// ---- DUTs/IO/Topology/Beckhoff_EPP1xxxEK1122_5ECABF39.TcDUT
{attribute 'GeneratedUsingTerminal: EK1122-0000-0018'}
{attribute addProperty BoxType "EK1122-0000-0018"}
{attribute addProperty Id "Beckhoff_EPP1xxxsub_EK1100EK1100_1FC0878B2A_0001_EPP1004_0061_0016EPP1004_D135F8DB8A_0002_EPP1008_0001_0016EPP1008_78E8D3DD12A_0003_EPP1008_0001_0017EPP1008_78E8D3DD12A_0004_EPP1008_0002_0016EPP1008_78E8D3DD12A_0005_EPP1008_0002_0017EPP1008_78E8D3DD12A_0006_EPP1008_0022_0016EPP1008_78E8D3DD12A_0007_EPP1018_0001_0016EPP1018_78E8D3DD12A_0008_EPP1018_0001_0017EPP1018_78E8D3DD12A_0009_EPP1018_0002_0016EPP1018_78E8D3DD12A_0010_EPP1018_0002_0017EPP1018_78E8D3DD12A_0011_EPP1111_0000_0016EPP1111_837A6B0314A_0012_EPP1111_0000_0017EPP1111_837A6B0314A_0013_EPP1111_0000_0018EPP1111_837A6B0314A_0014_EPP1258_0001_0016EPP1258_58F475DD56A_0015_EPP1258_0001_0017EPP1258_58F475DD56A_0016_EPP1258_0002_0016EPP1258_58F475DD56A_0017_EPP1258_0002_0017EPP1258_58F475DD56A_0018_EPP1321_0060_0016A_0018_EPP1321_0060_0016_F908F4F3378"}
{attribute addProperty CRC "1590345529"}
{attribute addProperty Size "762"}
{attribute addProperty Name "Beckhoff EPP1xxxEK1122"}
TYPE Beckhoff_EPP1xxxEK1122_5ECABF39 EXTENDS EK1122_1FC0878B :
STRUCT
	{attribute addProperty Name "Beckhoff EPP1xxxsub EK1100"}
	{attribute addProperty PreviousPort "Beckhoff EPP1xxxEK1122 : D"}
	Beckhoff_EPP1xxxsub_EK1100 : EK1100_1FC0878B;
	{attribute addProperty Name "A_0001(EPP1004-0061-0016)"}
	{attribute addProperty PreviousPort "Beckhoff EPP1xxxsub EK1100 : C"}
	A_0001_EPP1004_0061_0016 : EPP1004_D135F8DB;
	{attribute addProperty Name "A_0002(EPP1008-0001-0016)"}
	{attribute addProperty PreviousPort "A_0001(EPP1004-0061-0016) : B"}
	A_0002_EPP1008_0001_0016 : EPP1008_78E8D3DD;
	{attribute addProperty Name "A_0003(EPP1008-0001-0017)"}
	{attribute addProperty PreviousPort "A_0002(EPP1008-0001-0016) : B"}
	A_0003_EPP1008_0001_0017 : EPP1008_78E8D3DD;
	{attribute addProperty Name "A_0004(EPP1008-0002-0016)"}
	{attribute addProperty PreviousPort "A_0003(EPP1008-0001-0017) : B"}
	A_0004_EPP1008_0002_0016 : EPP1008_78E8D3DD;
	{attribute addProperty Name "A_0005(EPP1008-0002-0017)"}
	{attribute addProperty PreviousPort "A_0004(EPP1008-0002-0016) : B"}
	A_0005_EPP1008_0002_0017 : EPP1008_78E8D3DD;
	{attribute addProperty Name "A_0006(EPP1008-0022-0016)"}
	{attribute addProperty PreviousPort "A_0005(EPP1008-0002-0017) : B"}
	A_0006_EPP1008_0022_0016 : EPP1008_78E8D3DD;
	{attribute addProperty Name "A_0007(EPP1018-0001-0016)"}
	{attribute addProperty PreviousPort "A_0006(EPP1008-0022-0016) : B"}
	A_0007_EPP1018_0001_0016 : EPP1018_78E8D3DD;
	{attribute addProperty Name "A_0008(EPP1018-0001-0017)"}
	{attribute addProperty PreviousPort "A_0007(EPP1018-0001-0016) : B"}
	A_0008_EPP1018_0001_0017 : EPP1018_78E8D3DD;
	{attribute addProperty Name "A_0009(EPP1018-0002-0016)"}
	{attribute addProperty PreviousPort "A_0008(EPP1018-0001-0017) : B"}
	A_0009_EPP1018_0002_0016 : EPP1018_78E8D3DD;
	{attribute addProperty Name "A_0010(EPP1018-0002-0017)"}
	{attribute addProperty PreviousPort "A_0009(EPP1018-0002-0016) : B"}
	A_0010_EPP1018_0002_0017 : EPP1018_78E8D3DD;
	{attribute addProperty Name "A_0011(EPP1111-0000-0016)"}
	{attribute addProperty PreviousPort "A_0010(EPP1018-0002-0017) : B"}
	A_0011_EPP1111_0000_0016 : EPP1111_837A6B03;
	{attribute addProperty Name "A_0012(EPP1111-0000-0017)"}
	{attribute addProperty PreviousPort "A_0011(EPP1111-0000-0016) : B"}
	A_0012_EPP1111_0000_0017 : EPP1111_837A6B03;
	{attribute addProperty Name "A_0013(EPP1111-0000-0018)"}
	{attribute addProperty PreviousPort "A_0012(EPP1111-0000-0017) : B"}
	A_0013_EPP1111_0000_0018 : EPP1111_837A6B03;
	{attribute addProperty Name "A_0014(EPP1258-0001-0016)"}
	{attribute addProperty PreviousPort "A_0013(EPP1111-0000-0018) : B"}
	A_0014_EPP1258_0001_0016 : EPP1258_58F475DD;
	{attribute addProperty Name "A_0015(EPP1258-0001-0017)"}
	{attribute addProperty PreviousPort "A_0014(EPP1258-0001-0016) : B"}
	A_0015_EPP1258_0001_0017 : EPP1258_58F475DD;
	{attribute addProperty Name "A_0016(EPP1258-0002-0016)"}
	{attribute addProperty PreviousPort "A_0015(EPP1258-0001-0017) : B"}
	A_0016_EPP1258_0002_0016 : EPP1258_58F475DD;
	{attribute addProperty Name "A_0017(EPP1258-0002-0017)"}
	{attribute addProperty PreviousPort "A_0016(EPP1258-0002-0016) : B"}
	A_0017_EPP1258_0002_0017 : EPP1258_58F475DD;
	{attribute addProperty Name "A_0018(EPP1321-0060-0016)"}
	{attribute addProperty PreviousPort "A_0017(EPP1258-0002-0017) : B"}
	A_0018_EPP1321_0060_0016 : A_0018_EPP1321_0060_0016_F908F4F3;
END_STRUCT
END_TYPE

// ---- DUTs/IO/Topology/Beckhoff_EPP1xxx_3250354D.TcDUT
{attribute 'GeneratedUsingTerminal: EK1100-0000-0018'}
{attribute addProperty BoxType "EK1100-0000-0018"}
{attribute addProperty Id "Beckhoff_EPP1xxxEK1122Beckhoff_EPP1xxxEK1122_5ECABF39762"}
{attribute addProperty CRC "844117325"}
{attribute addProperty Size "762"}
{attribute addProperty Name "Beckhoff EPP1xxx"}
TYPE Beckhoff_EPP1xxx_3250354D EXTENDS EK1100_1FC0878B :
STRUCT
	{attribute addProperty Name "Beckhoff EPP1xxxEK1122"}
	{attribute addProperty PreviousPort "Beckhoff EPP1xxx : B"}
	Beckhoff_EPP1xxxEK1122 : Beckhoff_EPP1xxxEK1122_5ECABF39;
END_STRUCT
END_TYPE

// ---- DUTs/IO/Topology/Beckhoff_EPP2xxxEK1122_56176A05.TcDUT
{attribute 'GeneratedUsingTerminal: EK1122-0000-0018'}
{attribute addProperty BoxType "EK1122-0000-0018"}
{attribute addProperty Id "Beckhoff_EPP2xxxsub_EK1100EK1100_1FC0878B2A_0001_EPP2008_0001_0016EPP2008_E2806B9511A_0002_EPP2008_0001_0017EPP2008_E2806B9511A_0003_EPP2008_0001_0018EPP2008_E2806B9511A_0004_EPP2008_0002_0016EPP2008_E2806B9511A_0005_EPP2008_0002_0017EPP2008_E2806B9511A_0006_EPP2008_0002_0018EPP2008_E2806B9511A_0007_EPP2008_0022_0016EPP2008_E2806B9511A_0008_EPP2028_0001_0016EPP2028_E2806B9511A_0009_EPP2028_0001_0017EPP2028_E2806B9511A_0010_EPP2028_0002_0016EPP2028_E2806B9511A_0011_EPP2028_0002_0017EPP2028_E2806B9511A_0012_EPP2038_0001_0016EPP2038_3AE10DD720A_0013_EPP2038_0002_0016EPP2038_3AE10DD720A_0014_EPP2304_0061_0016EPP2304_473048998A_0015_EPP2304_0061_0017EPP2304_473048998A_0016_EPP2304_0061_0018EPP2304_473048998A_0017_EPP2308_0001_0016EPP2308_F6D9A8D112A_0018_EPP2308_0001_0017EPP2308_F6D9A8D112A_0019_EPP2308_0001_0018EPP2308_F6D9A8D112A_0020_EPP2308_0002_0016EPP2308_F6D9A8D112A_0021_EPP2308_0002_0017EPP2308_F6D9A8D112A_0022_EPP2308_0002_0018EPP2308_F6D9A8D112A_0023_EPP2316_0003_0016EPP2316_CAC4656D44A_0024_EPP2316_0003_0017EPP2316_CAC4656D44A_0025_EPP2316_0003_0018EPP2316_D286688344A_0026_EPP2316_0008_0016EPP2316_CAC4656D44A_0027_EPP2316_0008_0017EPP2316_CAC4656D44A_0028_EPP2316_0008_0018EPP2316_D286688344A_0029_EPP2318_0001_0016EPP2318_F6D9A8D112A_0030_EPP2318_0001_0017EPP2318_F6D9A8D112A_0031_EPP2318_0001_0018EPP2318_F6D9A8D112A_0032_EPP2318_0002_0016EPP2318_F6D9A8D112A_0033_EPP2318_0002_0017EPP2318_F6D9A8D112A_0034_EPP2318_0002_0018EPP2318_F6D9A8D112A_0035_EPP2328_0001_0016EPP2328_F6D9A8D112A_0036_EPP2328_0001_0017EPP2328_F6D9A8D112A_0037_EPP2328_0001_0018EPP2328_F6D9A8D112A_0038_EPP2328_0002_0016EPP2328_F6D9A8D112A_0039_EPP2328_0002_0017EPP2328_F6D9A8D112A_0040_EPP2328_0002_0018EPP2328_F6D9A8D112A_0041_EPP2334_0061_0016EPP2334_F6D9A8D112A_0042_EPP2334_0061_0017EPP2334_F6D9A8D112A_0043_EPP2334_0061_0018EPP2334_F6D9A8D112A_0044_EPP2334_0061_0019EPP2334_F6D9A8D112A_0045_EPP2338_0001_0016EPP2338_7699BCF620A_0046_EPP2338_0001_0017EPP2338_7699BCF620A_0047_EPP2338_0001_0018EPP2338_7699BCF620A_0048_EPP2338_0002_0016EPP2338_7699BCF620A_0049_EPP2338_0002_0017EPP2338_7699BCF620A_0050_EPP2338_0002_0018EPP2338_7699BCF620A_0051_EPP2338_1001_0017EPP2338_7699BCF620A_0052_EPP2338_1001_0018EPP2338_7699BCF620A_0053_EPP2338_1001_0019EPP2338_7699BCF620A_0054_EPP2338_1002_0017EPP2338_7699BCF620A_0055_EPP2338_1002_0018EPP2338_7699BCF620A_0056_EPP2338_1002_0019EPP2338_7699BCF620A_0057_EPP2339_0003_0016EPP2339_B2B612E850A_0058_EPP2339_0021_0016EPP2339_8DFD155836A_0059_EPP2339_0021_0017EPP2339_4CF33DED36A_0060_EPP2339_0021_0018EPP2339_4CF33DED36A_0061_EPP2339_0022_0016EPP2339_8DFD155836A_0062_EPP2339_0022_0017EPP2339_4CF33DED36A_0063_EPP2339_0022_0018EPP2339_4CF33DED36A_0064_EPP2349_0021_0016EPP2349_8DFD155836A_0065_EPP2349_0021_0017EPP2349_4CF33DED36A_0066_EPP2349_0021_0018EPP2349_4CF33DED36A_0067_EPP2349_0022_0016EPP2349_8DFD155836A_0068_EPP2349_0022_0017EPP2349_4CF33DED36A_0069_EPP2349_0022_0018EPP2349_4CF33DED36A_0070_EPP2624_0002_0016EPP2624_7B64371E7A_0071_EPP2809_0021_0016EPP2809_2B6483BD19A_0072_EPP2809_0022_0016EPP2809_2B6483BD19A_0073_EPP2816_0004_0016EPP2816_F9F6AB8251A_0074_EPP2816_0004_0017EPP2816_F9F6AB8251A_0075_EPP2816_0008_0016EPP2816_0129644951A_0076_EPP2816_0008_0017EPP2816_0129644951A_0077_EPP2816_0008_0018EPP2816_0129644951A_0078_EPP2816_0010_0016EPP2816_0129644951A_0079_EPP2816_0010_0017EPP2816_0129644951A_0080_EPP2816_0010_0018EPP2816_0129644951A_0081_EPP2817_0008_0016EPP2817_7CB3CE2970A_0082_EPP2817_0008_0017EPP2817_7CB3CE2970A_0083_EPP2817_0008_0018EPP2817_7CB3CE2970"}
{attribute addProperty CRC "1444375045"}
{attribute addProperty Size "2100"}
{attribute addProperty Name "Beckhoff EPP2xxxEK1122"}
TYPE Beckhoff_EPP2xxxEK1122_56176A05 EXTENDS EK1122_1FC0878B :
STRUCT
	{attribute addProperty Name "Beckhoff EPP2xxxsub EK1100"}
	{attribute addProperty PreviousPort "Beckhoff EPP2xxxEK1122 : D"}
	Beckhoff_EPP2xxxsub_EK1100 : EK1100_1FC0878B;
	{attribute addProperty Name "A_0001(EPP2008-0001-0016)"}
	{attribute addProperty PreviousPort "Beckhoff EPP2xxxsub EK1100 : C"}
	A_0001_EPP2008_0001_0016 : EPP2008_E2806B95;
	{attribute addProperty Name "A_0002(EPP2008-0001-0017)"}
	{attribute addProperty PreviousPort "A_0001(EPP2008-0001-0016) : B"}
	A_0002_EPP2008_0001_0017 : EPP2008_E2806B95;
	{attribute addProperty Name "A_0003(EPP2008-0001-0018)"}
	{attribute addProperty PreviousPort "A_0002(EPP2008-0001-0017) : B"}
	A_0003_EPP2008_0001_0018 : EPP2008_E2806B95;
	{attribute addProperty Name "A_0004(EPP2008-0002-0016)"}
	{attribute addProperty PreviousPort "A_0003(EPP2008-0001-0018) : B"}
	A_0004_EPP2008_0002_0016 : EPP2008_E2806B95;
	{attribute addProperty Name "A_0005(EPP2008-0002-0017)"}
	{attribute addProperty PreviousPort "A_0004(EPP2008-0002-0016) : B"}
	A_0005_EPP2008_0002_0017 : EPP2008_E2806B95;
	{attribute addProperty Name "A_0006(EPP2008-0002-0018)"}
	{attribute addProperty PreviousPort "A_0005(EPP2008-0002-0017) : B"}
	A_0006_EPP2008_0002_0018 : EPP2008_E2806B95;
	{attribute addProperty Name "A_0007(EPP2008-0022-0016)"}
	{attribute addProperty PreviousPort "A_0006(EPP2008-0002-0018) : B"}
	A_0007_EPP2008_0022_0016 : EPP2008_E2806B95;
	{attribute addProperty Name "A_0008(EPP2028-0001-0016)"}
	{attribute addProperty PreviousPort "A_0007(EPP2008-0022-0016) : B"}
	A_0008_EPP2028_0001_0016 : EPP2028_E2806B95;
	{attribute addProperty Name "A_0009(EPP2028-0001-0017)"}
	{attribute addProperty PreviousPort "A_0008(EPP2028-0001-0016) : B"}
	A_0009_EPP2028_0001_0017 : EPP2028_E2806B95;
	{attribute addProperty Name "A_0010(EPP2028-0002-0016)"}
	{attribute addProperty PreviousPort "A_0009(EPP2028-0001-0017) : B"}
	A_0010_EPP2028_0002_0016 : EPP2028_E2806B95;
	{attribute addProperty Name "A_0011(EPP2028-0002-0017)"}
	{attribute addProperty PreviousPort "A_0010(EPP2028-0002-0016) : B"}
	A_0011_EPP2028_0002_0017 : EPP2028_E2806B95;
	{attribute addProperty Name "A_0012(EPP2038-0001-0016)"}
	{attribute addProperty PreviousPort "A_0011(EPP2028-0002-0017) : B"}
	A_0012_EPP2038_0001_0016 : EPP2038_3AE10DD7;
	{attribute addProperty Name "A_0013(EPP2038-0002-0016)"}
	{attribute addProperty PreviousPort "A_0012(EPP2038-0001-0016) : B"}
	A_0013_EPP2038_0002_0016 : EPP2038_3AE10DD7;
	{attribute addProperty Name "A_0014(EPP2304-0061-0016)"}
	{attribute addProperty PreviousPort "A_0013(EPP2038-0002-0016) : B"}
	A_0014_EPP2304_0061_0016 : EPP2304_47304899;
	{attribute addProperty Name "A_0015(EPP2304-0061-0017)"}
	{attribute addProperty PreviousPort "A_0014(EPP2304-0061-0016) : B"}
	A_0015_EPP2304_0061_0017 : EPP2304_47304899;
	{attribute addProperty Name "A_0016(EPP2304-0061-0018)"}
	{attribute addProperty PreviousPort "A_0015(EPP2304-0061-0017) : B"}
	A_0016_EPP2304_0061_0018 : EPP2304_47304899;
	{attribute addProperty Name "A_0017(EPP2308-0001-0016)"}
	{attribute addProperty PreviousPort "A_0016(EPP2304-0061-0018) : B"}
	A_0017_EPP2308_0001_0016 : EPP2308_F6D9A8D1;
	{attribute addProperty Name "A_0018(EPP2308-0001-0017)"}
	{attribute addProperty PreviousPort "A_0017(EPP2308-0001-0016) : B"}
	A_0018_EPP2308_0001_0017 : EPP2308_F6D9A8D1;
	{attribute addProperty Name "A_0019(EPP2308-0001-0018)"}
	{attribute addProperty PreviousPort "A_0018(EPP2308-0001-0017) : B"}
	A_0019_EPP2308_0001_0018 : EPP2308_F6D9A8D1;
	{attribute addProperty Name "A_0020(EPP2308-0002-0016)"}
	{attribute addProperty PreviousPort "A_0019(EPP2308-0001-0018) : B"}
	A_0020_EPP2308_0002_0016 : EPP2308_F6D9A8D1;
	{attribute addProperty Name "A_0021(EPP2308-0002-0017)"}
	{attribute addProperty PreviousPort "A_0020(EPP2308-0002-0016) : B"}
	A_0021_EPP2308_0002_0017 : EPP2308_F6D9A8D1;
	{attribute addProperty Name "A_0022(EPP2308-0002-0018)"}
	{attribute addProperty PreviousPort "A_0021(EPP2308-0002-0017) : B"}
	A_0022_EPP2308_0002_0018 : EPP2308_F6D9A8D1;
	{attribute addProperty Name "A_0023(EPP2316-0003-0016)"}
	{attribute addProperty PreviousPort "A_0022(EPP2308-0002-0018) : B"}
	A_0023_EPP2316_0003_0016 : EPP2316_CAC4656D;
	{attribute addProperty Name "A_0024(EPP2316-0003-0017)"}
	{attribute addProperty PreviousPort "A_0023(EPP2316-0003-0016) : B"}
	A_0024_EPP2316_0003_0017 : EPP2316_CAC4656D;
	{attribute addProperty Name "A_0025(EPP2316-0003-0018)"}
	{attribute addProperty PreviousPort "A_0024(EPP2316-0003-0017) : B"}
	A_0025_EPP2316_0003_0018 : EPP2316_D2866883;
	{attribute addProperty Name "A_0026(EPP2316-0008-0016)"}
	{attribute addProperty PreviousPort "A_0025(EPP2316-0003-0018) : B"}
	A_0026_EPP2316_0008_0016 : EPP2316_CAC4656D;
	{attribute addProperty Name "A_0027(EPP2316-0008-0017)"}
	{attribute addProperty PreviousPort "A_0026(EPP2316-0008-0016) : B"}
	A_0027_EPP2316_0008_0017 : EPP2316_CAC4656D;
	{attribute addProperty Name "A_0028(EPP2316-0008-0018)"}
	{attribute addProperty PreviousPort "A_0027(EPP2316-0008-0017) : B"}
	A_0028_EPP2316_0008_0018 : EPP2316_D2866883;
	{attribute addProperty Name "A_0029(EPP2318-0001-0016)"}
	{attribute addProperty PreviousPort "A_0028(EPP2316-0008-0018) : B"}
	A_0029_EPP2318_0001_0016 : EPP2318_F6D9A8D1;
	{attribute addProperty Name "A_0030(EPP2318-0001-0017)"}
	{attribute addProperty PreviousPort "A_0029(EPP2318-0001-0016) : B"}
	A_0030_EPP2318_0001_0017 : EPP2318_F6D9A8D1;
	{attribute addProperty Name "A_0031(EPP2318-0001-0018)"}
	{attribute addProperty PreviousPort "A_0030(EPP2318-0001-0017) : B"}
	A_0031_EPP2318_0001_0018 : EPP2318_F6D9A8D1;
	{attribute addProperty Name "A_0032(EPP2318-0002-0016)"}
	{attribute addProperty PreviousPort "A_0031(EPP2318-0001-0018) : B"}
	A_0032_EPP2318_0002_0016 : EPP2318_F6D9A8D1;
	{attribute addProperty Name "A_0033(EPP2318-0002-0017)"}
	{attribute addProperty PreviousPort "A_0032(EPP2318-0002-0016) : B"}
	A_0033_EPP2318_0002_0017 : EPP2318_F6D9A8D1;
	{attribute addProperty Name "A_0034(EPP2318-0002-0018)"}
	{attribute addProperty PreviousPort "A_0033(EPP2318-0002-0017) : B"}
	A_0034_EPP2318_0002_0018 : EPP2318_F6D9A8D1;
	{attribute addProperty Name "A_0035(EPP2328-0001-0016)"}
	{attribute addProperty PreviousPort "A_0034(EPP2318-0002-0018) : B"}
	A_0035_EPP2328_0001_0016 : EPP2328_F6D9A8D1;
	{attribute addProperty Name "A_0036(EPP2328-0001-0017)"}
	{attribute addProperty PreviousPort "A_0035(EPP2328-0001-0016) : B"}
	A_0036_EPP2328_0001_0017 : EPP2328_F6D9A8D1;
	{attribute addProperty Name "A_0037(EPP2328-0001-0018)"}
	{attribute addProperty PreviousPort "A_0036(EPP2328-0001-0017) : B"}
	A_0037_EPP2328_0001_0018 : EPP2328_F6D9A8D1;
	{attribute addProperty Name "A_0038(EPP2328-0002-0016)"}
	{attribute addProperty PreviousPort "A_0037(EPP2328-0001-0018) : B"}
	A_0038_EPP2328_0002_0016 : EPP2328_F6D9A8D1;
	{attribute addProperty Name "A_0039(EPP2328-0002-0017)"}
	{attribute addProperty PreviousPort "A_0038(EPP2328-0002-0016) : B"}
	A_0039_EPP2328_0002_0017 : EPP2328_F6D9A8D1;
	{attribute addProperty Name "A_0040(EPP2328-0002-0018)"}
	{attribute addProperty PreviousPort "A_0039(EPP2328-0002-0017) : B"}
	A_0040_EPP2328_0002_0018 : EPP2328_F6D9A8D1;
	{attribute addProperty Name "A_0041(EPP2334-0061-0016)"}
	{attribute addProperty PreviousPort "A_0040(EPP2328-0002-0018) : B"}
	A_0041_EPP2334_0061_0016 : EPP2334_F6D9A8D1;
	{attribute addProperty Name "A_0042(EPP2334-0061-0017)"}
	{attribute addProperty PreviousPort "A_0041(EPP2334-0061-0016) : B"}
	A_0042_EPP2334_0061_0017 : EPP2334_F6D9A8D1;
	{attribute addProperty Name "A_0043(EPP2334-0061-0018)"}
	{attribute addProperty PreviousPort "A_0042(EPP2334-0061-0017) : B"}
	A_0043_EPP2334_0061_0018 : EPP2334_F6D9A8D1;
	{attribute addProperty Name "A_0044(EPP2334-0061-0019)"}
	{attribute addProperty PreviousPort "A_0043(EPP2334-0061-0018) : B"}
	A_0044_EPP2334_0061_0019 : EPP2334_F6D9A8D1;
	{attribute addProperty Name "A_0045(EPP2338-0001-0016)"}
	{attribute addProperty PreviousPort "A_0044(EPP2334-0061-0019) : B"}
	A_0045_EPP2338_0001_0016 : EPP2338_7699BCF6;
	{attribute addProperty Name "A_0046(EPP2338-0001-0017)"}
	{attribute addProperty PreviousPort "A_0045(EPP2338-0001-0016) : B"}
	A_0046_EPP2338_0001_0017 : EPP2338_7699BCF6;
	{attribute addProperty Name "A_0047(EPP2338-0001-0018)"}
	{attribute addProperty PreviousPort "A_0046(EPP2338-0001-0017) : B"}
	A_0047_EPP2338_0001_0018 : EPP2338_7699BCF6;
	{attribute addProperty Name "A_0048(EPP2338-0002-0016)"}
	{attribute addProperty PreviousPort "A_0047(EPP2338-0001-0018) : B"}
	A_0048_EPP2338_0002_0016 : EPP2338_7699BCF6;
	{attribute addProperty Name "A_0049(EPP2338-0002-0017)"}
	{attribute addProperty PreviousPort "A_0048(EPP2338-0002-0016) : B"}
	A_0049_EPP2338_0002_0017 : EPP2338_7699BCF6;
	{attribute addProperty Name "A_0050(EPP2338-0002-0018)"}
	{attribute addProperty PreviousPort "A_0049(EPP2338-0002-0017) : B"}
	A_0050_EPP2338_0002_0018 : EPP2338_7699BCF6;
	{attribute addProperty Name "A_0051(EPP2338-1001-0017)"}
	{attribute addProperty PreviousPort "A_0050(EPP2338-0002-0018) : B"}
	A_0051_EPP2338_1001_0017 : EPP2338_7699BCF6;
	{attribute addProperty Name "A_0052(EPP2338-1001-0018)"}
	{attribute addProperty PreviousPort "A_0051(EPP2338-1001-0017) : B"}
	A_0052_EPP2338_1001_0018 : EPP2338_7699BCF6;
	{attribute addProperty Name "A_0053(EPP2338-1001-0019)"}
	{attribute addProperty PreviousPort "A_0052(EPP2338-1001-0018) : B"}
	A_0053_EPP2338_1001_0019 : EPP2338_7699BCF6;
	{attribute addProperty Name "A_0054(EPP2338-1002-0017)"}
	{attribute addProperty PreviousPort "A_0053(EPP2338-1001-0019) : B"}
	A_0054_EPP2338_1002_0017 : EPP2338_7699BCF6;
	{attribute addProperty Name "A_0055(EPP2338-1002-0018)"}
	{attribute addProperty PreviousPort "A_0054(EPP2338-1002-0017) : B"}
	A_0055_EPP2338_1002_0018 : EPP2338_7699BCF6;
	{attribute addProperty Name "A_0056(EPP2338-1002-0019)"}
	{attribute addProperty PreviousPort "A_0055(EPP2338-1002-0018) : B"}
	A_0056_EPP2338_1002_0019 : EPP2338_7699BCF6;
	{attribute addProperty Name "A_0057(EPP2339-0003-0016)"}
	{attribute addProperty PreviousPort "A_0056(EPP2338-1002-0019) : B"}
	A_0057_EPP2339_0003_0016 : EPP2339_B2B612E8;
	{attribute addProperty Name "A_0058(EPP2339-0021-0016)"}
	{attribute addProperty PreviousPort "A_0057(EPP2339-0003-0016) : B"}
	A_0058_EPP2339_0021_0016 : EPP2339_8DFD1558;
	{attribute addProperty Name "A_0059(EPP2339-0021-0017)"}
	{attribute addProperty PreviousPort "A_0058(EPP2339-0021-0016) : B"}
	A_0059_EPP2339_0021_0017 : EPP2339_4CF33DED;
	{attribute addProperty Name "A_0060(EPP2339-0021-0018)"}
	{attribute addProperty PreviousPort "A_0059(EPP2339-0021-0017) : B"}
	A_0060_EPP2339_0021_0018 : EPP2339_4CF33DED;
	{attribute addProperty Name "A_0061(EPP2339-0022-0016)"}
	{attribute addProperty PreviousPort "A_0060(EPP2339-0021-0018) : B"}
	A_0061_EPP2339_0022_0016 : EPP2339_8DFD1558;
	{attribute addProperty Name "A_0062(EPP2339-0022-0017)"}
	{attribute addProperty PreviousPort "A_0061(EPP2339-0022-0016) : B"}
	A_0062_EPP2339_0022_0017 : EPP2339_4CF33DED;
	{attribute addProperty Name "A_0063(EPP2339-0022-0018)"}
	{attribute addProperty PreviousPort "A_0062(EPP2339-0022-0017) : B"}
	A_0063_EPP2339_0022_0018 : EPP2339_4CF33DED;
	{attribute addProperty Name "A_0064(EPP2349-0021-0016)"}
	{attribute addProperty PreviousPort "A_0063(EPP2339-0022-0018) : B"}
	A_0064_EPP2349_0021_0016 : EPP2349_8DFD1558;
	{attribute addProperty Name "A_0065(EPP2349-0021-0017)"}
	{attribute addProperty PreviousPort "A_0064(EPP2349-0021-0016) : B"}
	A_0065_EPP2349_0021_0017 : EPP2349_4CF33DED;
	{attribute addProperty Name "A_0066(EPP2349-0021-0018)"}
	{attribute addProperty PreviousPort "A_0065(EPP2349-0021-0017) : B"}
	A_0066_EPP2349_0021_0018 : EPP2349_4CF33DED;
	{attribute addProperty Name "A_0067(EPP2349-0022-0016)"}
	{attribute addProperty PreviousPort "A_0066(EPP2349-0021-0018) : B"}
	A_0067_EPP2349_0022_0016 : EPP2349_8DFD1558;
	{attribute addProperty Name "A_0068(EPP2349-0022-0017)"}
	{attribute addProperty PreviousPort "A_0067(EPP2349-0022-0016) : B"}
	A_0068_EPP2349_0022_0017 : EPP2349_4CF33DED;
	{attribute addProperty Name "A_0069(EPP2349-0022-0018)"}
	{attribute addProperty PreviousPort "A_0068(EPP2349-0022-0017) : B"}
	A_0069_EPP2349_0022_0018 : EPP2349_4CF33DED;
	{attribute addProperty Name "A_0070(EPP2624-0002-0016)"}
	{attribute addProperty PreviousPort "A_0069(EPP2349-0022-0018) : B"}
	A_0070_EPP2624_0002_0016 : EPP2624_7B64371E;
	{attribute addProperty Name "A_0071(EPP2809-0021-0016)"}
	{attribute addProperty PreviousPort "A_0070(EPP2624-0002-0016) : B"}
	A_0071_EPP2809_0021_0016 : EPP2809_2B6483BD;
	{attribute addProperty Name "A_0072(EPP2809-0022-0016)"}
	{attribute addProperty PreviousPort "A_0071(EPP2809-0021-0016) : B"}
	A_0072_EPP2809_0022_0016 : EPP2809_2B6483BD;
	{attribute addProperty Name "A_0073(EPP2816-0004-0016)"}
	{attribute addProperty PreviousPort "A_0072(EPP2809-0022-0016) : B"}
	A_0073_EPP2816_0004_0016 : EPP2816_F9F6AB82;
	{attribute addProperty Name "A_0074(EPP2816-0004-0017)"}
	{attribute addProperty PreviousPort "A_0073(EPP2816-0004-0016) : B"}
	A_0074_EPP2816_0004_0017 : EPP2816_F9F6AB82;
	{attribute addProperty Name "A_0075(EPP2816-0008-0016)"}
	{attribute addProperty PreviousPort "A_0074(EPP2816-0004-0017) : B"}
	A_0075_EPP2816_0008_0016 : EPP2816_01296449;
	{attribute addProperty Name "A_0076(EPP2816-0008-0017)"}
	{attribute addProperty PreviousPort "A_0075(EPP2816-0008-0016) : B"}
	A_0076_EPP2816_0008_0017 : EPP2816_01296449;
	{attribute addProperty Name "A_0077(EPP2816-0008-0018)"}
	{attribute addProperty PreviousPort "A_0076(EPP2816-0008-0017) : B"}
	A_0077_EPP2816_0008_0018 : EPP2816_01296449;
	{attribute addProperty Name "A_0078(EPP2816-0010-0016)"}
	{attribute addProperty PreviousPort "A_0077(EPP2816-0008-0018) : B"}
	A_0078_EPP2816_0010_0016 : EPP2816_01296449;
	{attribute addProperty Name "A_0079(EPP2816-0010-0017)"}
	{attribute addProperty PreviousPort "A_0078(EPP2816-0010-0016) : B"}
	A_0079_EPP2816_0010_0017 : EPP2816_01296449;
	{attribute addProperty Name "A_0080(EPP2816-0010-0018)"}
	{attribute addProperty PreviousPort "A_0079(EPP2816-0010-0017) : B"}
	A_0080_EPP2816_0010_0018 : EPP2816_01296449;
	{attribute addProperty Name "A_0081(EPP2817-0008-0016)"}
	{attribute addProperty PreviousPort "A_0080(EPP2816-0010-0018) : B"}
	A_0081_EPP2817_0008_0016 : EPP2817_7CB3CE29;
	{attribute addProperty Name "A_0082(EPP2817-0008-0017)"}
	{attribute addProperty PreviousPort "A_0081(EPP2817-0008-0016) : B"}
	A_0082_EPP2817_0008_0017 : EPP2817_7CB3CE29;
	{attribute addProperty Name "A_0083(EPP2817-0008-0018)"}
	{attribute addProperty PreviousPort "A_0082(EPP2817-0008-0017) : B"}
	A_0083_EPP2817_0008_0018 : EPP2817_7CB3CE29;
END_STRUCT
END_TYPE

// ---- DUTs/IO/Topology/Beckhoff_EPP2xxx_8ED37E64.TcDUT
{attribute 'GeneratedUsingTerminal: EK1100-0000-0018'}
{attribute addProperty BoxType "EK1100-0000-0018"}
{attribute addProperty Id "Beckhoff_EPP2xxxEK1122Beckhoff_EPP2xxxEK1122_56176A052100"}
{attribute addProperty CRC "2396225124"}
{attribute addProperty Size "2100"}
{attribute addProperty Name "Beckhoff EPP2xxx"}
TYPE Beckhoff_EPP2xxx_8ED37E64 EXTENDS EK1100_1FC0878B :
STRUCT
	{attribute addProperty Name "Beckhoff EPP2xxxEK1122"}
	{attribute addProperty PreviousPort "Beckhoff EPP2xxx : B"}
	Beckhoff_EPP2xxxEK1122 : Beckhoff_EPP2xxxEK1122_56176A05;
END_STRUCT
END_TYPE

// ---- DUTs/IO/Topology/Beckhoff_EPP3xxxEK1122_A76E71A7.TcDUT
{attribute 'GeneratedUsingTerminal: EK1122-0000-0018'}
{attribute addProperty BoxType "EK1122-0000-0018"}
{attribute addProperty Id "Beckhoff_EPP3xxxsub_EK1100EK1100_1FC0878B2A_0001_EPP3174_0002_0016EPP3174_DCC7866252A_0002_EPP3174_0002_0017EPP3174_DCC7866252A_0003_EPP3174_0002_0018EPP3174_DCC7866252A_0004_EPP3184_0002_0016EPP3184_DCC7866252A_0005_EPP3184_0002_0017EPP3184_DCC7866252A_0006_EPP3184_0002_0018EPP3184_DCC7866252A_0007_EPP3184_0002_0019EPP3184_DCC7866252A_0008_EPP3204_0002_0016EPP3204_6CD7E11952A_0009_EPP3204_0002_0017EPP3204_AB25C3AC48A_0010_EPP3204_0002_0018EPP3204_AB25C3AC48A_0011_EPP3204_0002_0019EPP3204_AB25C3AC48A_0012_EPP3314_0002_0016EPP3314_E65CDB1C48A_0013_EPP3314_0002_0017EPP3314_E65CDB1C48A_0014_EPP3314_0002_0018EPP3314_E65CDB1C48A_0015_EPP3632_0001_0016EPP3632_E2B98A5C86A_0016_EPP3632_0001_0017EPP3632_E2B98A5C86A_0017_EPP3744_0041_0016EPP3744_315C92D470A_0018_EPP3744_0041_0017EPP3744_315C92D470A_0019_EPP3744_0041_0018EPP3744_315C92D470A_0020_EPP3744_1041_0016EPP3744_315C92D470A_0021_EPP3744_1041_0017EPP3744_315C92D470A_0022_EPP3744_1041_0018EPP3744_315C92D470A_0023_EPP3744_1041_0019EPP3744_315C92D470A_0024_EPP3744_1041_0020EPP3744_315C92D470A_0025_EPP3752_0000_0017EPP3752_C992DA1B42"}
{attribute addProperty CRC "2809033127"}
{attribute addProperty Size "1480"}
{attribute addProperty Name "Beckhoff EPP3xxxEK1122"}
TYPE Beckhoff_EPP3xxxEK1122_A76E71A7 EXTENDS EK1122_1FC0878B :
STRUCT
	{attribute addProperty Name "Beckhoff EPP3xxxsub EK1100"}
	{attribute addProperty PreviousPort "Beckhoff EPP3xxxEK1122 : D"}
	Beckhoff_EPP3xxxsub_EK1100 : EK1100_1FC0878B;
	{attribute addProperty Name "A_0001(EPP3174-0002-0016)"}
	{attribute addProperty PreviousPort "Beckhoff EPP3xxxsub EK1100 : C"}
	A_0001_EPP3174_0002_0016 : EPP3174_DCC78662;
	{attribute addProperty Name "A_0002(EPP3174-0002-0017)"}
	{attribute addProperty PreviousPort "A_0001(EPP3174-0002-0016) : B"}
	A_0002_EPP3174_0002_0017 : EPP3174_DCC78662;
	{attribute addProperty Name "A_0003(EPP3174-0002-0018)"}
	{attribute addProperty PreviousPort "A_0002(EPP3174-0002-0017) : B"}
	A_0003_EPP3174_0002_0018 : EPP3174_DCC78662;
	{attribute addProperty Name "A_0004(EPP3184-0002-0016)"}
	{attribute addProperty PreviousPort "A_0003(EPP3174-0002-0018) : B"}
	A_0004_EPP3184_0002_0016 : EPP3184_DCC78662;
	{attribute addProperty Name "A_0005(EPP3184-0002-0017)"}
	{attribute addProperty PreviousPort "A_0004(EPP3184-0002-0016) : B"}
	A_0005_EPP3184_0002_0017 : EPP3184_DCC78662;
	{attribute addProperty Name "A_0006(EPP3184-0002-0018)"}
	{attribute addProperty PreviousPort "A_0005(EPP3184-0002-0017) : B"}
	A_0006_EPP3184_0002_0018 : EPP3184_DCC78662;
	{attribute addProperty Name "A_0007(EPP3184-0002-0019)"}
	{attribute addProperty PreviousPort "A_0006(EPP3184-0002-0018) : B"}
	A_0007_EPP3184_0002_0019 : EPP3184_DCC78662;
	{attribute addProperty Name "A_0008(EPP3204-0002-0016)"}
	{attribute addProperty PreviousPort "A_0007(EPP3184-0002-0019) : B"}
	A_0008_EPP3204_0002_0016 : EPP3204_6CD7E119;
	{attribute addProperty Name "A_0009(EPP3204-0002-0017)"}
	{attribute addProperty PreviousPort "A_0008(EPP3204-0002-0016) : B"}
	A_0009_EPP3204_0002_0017 : EPP3204_AB25C3AC;
	{attribute addProperty Name "A_0010(EPP3204-0002-0018)"}
	{attribute addProperty PreviousPort "A_0009(EPP3204-0002-0017) : B"}
	A_0010_EPP3204_0002_0018 : EPP3204_AB25C3AC;
	{attribute addProperty Name "A_0011(EPP3204-0002-0019)"}
	{attribute addProperty PreviousPort "A_0010(EPP3204-0002-0018) : B"}
	A_0011_EPP3204_0002_0019 : EPP3204_AB25C3AC;
	{attribute addProperty Name "A_0012(EPP3314-0002-0016)"}
	{attribute addProperty PreviousPort "A_0011(EPP3204-0002-0019) : B"}
	A_0012_EPP3314_0002_0016 : EPP3314_E65CDB1C;
	{attribute addProperty Name "A_0013(EPP3314-0002-0017)"}
	{attribute addProperty PreviousPort "A_0012(EPP3314-0002-0016) : B"}
	A_0013_EPP3314_0002_0017 : EPP3314_E65CDB1C;
	{attribute addProperty Name "A_0014(EPP3314-0002-0018)"}
	{attribute addProperty PreviousPort "A_0013(EPP3314-0002-0017) : B"}
	A_0014_EPP3314_0002_0018 : EPP3314_E65CDB1C;
	{attribute addProperty Name "A_0015(EPP3632-0001-0016)"}
	{attribute addProperty PreviousPort "A_0014(EPP3314-0002-0018) : B"}
	A_0015_EPP3632_0001_0016 : EPP3632_E2B98A5C;
	{attribute addProperty Name "A_0016(EPP3632-0001-0017)"}
	{attribute addProperty PreviousPort "A_0015(EPP3632-0001-0016) : B"}
	A_0016_EPP3632_0001_0017 : EPP3632_E2B98A5C;
	{attribute addProperty Name "A_0017(EPP3744-0041-0016)"}
	{attribute addProperty PreviousPort "A_0016(EPP3632-0001-0017) : B"}
	A_0017_EPP3744_0041_0016 : EPP3744_315C92D4;
	{attribute addProperty Name "A_0018(EPP3744-0041-0017)"}
	{attribute addProperty PreviousPort "A_0017(EPP3744-0041-0016) : B"}
	A_0018_EPP3744_0041_0017 : EPP3744_315C92D4;
	{attribute addProperty Name "A_0019(EPP3744-0041-0018)"}
	{attribute addProperty PreviousPort "A_0018(EPP3744-0041-0017) : B"}
	A_0019_EPP3744_0041_0018 : EPP3744_315C92D4;
	{attribute addProperty Name "A_0020(EPP3744-1041-0016)"}
	{attribute addProperty PreviousPort "A_0019(EPP3744-0041-0018) : B"}
	A_0020_EPP3744_1041_0016 : EPP3744_315C92D4;
	{attribute addProperty Name "A_0021(EPP3744-1041-0017)"}
	{attribute addProperty PreviousPort "A_0020(EPP3744-1041-0016) : B"}
	A_0021_EPP3744_1041_0017 : EPP3744_315C92D4;
	{attribute addProperty Name "A_0022(EPP3744-1041-0018)"}
	{attribute addProperty PreviousPort "A_0021(EPP3744-1041-0017) : B"}
	A_0022_EPP3744_1041_0018 : EPP3744_315C92D4;
	{attribute addProperty Name "A_0023(EPP3744-1041-0019)"}
	{attribute addProperty PreviousPort "A_0022(EPP3744-1041-0018) : B"}
	A_0023_EPP3744_1041_0019 : EPP3744_315C92D4;
	{attribute addProperty Name "A_0024(EPP3744-1041-0020)"}
	{attribute addProperty PreviousPort "A_0023(EPP3744-1041-0019) : B"}
	A_0024_EPP3744_1041_0020 : EPP3744_315C92D4;
	{attribute addProperty Name "A_0025(EPP3752-0000-0017)"}
	{attribute addProperty PreviousPort "A_0024(EPP3744-1041-0020) : B"}
	A_0025_EPP3752_0000_0017 : EPP3752_C992DA1B;
END_STRUCT
END_TYPE

// ---- DUTs/IO/Topology/Beckhoff_EPP3xxx_37FEE8A0.TcDUT
{attribute 'GeneratedUsingTerminal: EK1100-0000-0018'}
{attribute addProperty BoxType "EK1100-0000-0018"}
{attribute addProperty Id "Beckhoff_EPP3xxxEK1122Beckhoff_EPP3xxxEK1122_A76E71A71480"}
{attribute addProperty CRC "939452576"}
{attribute addProperty Size "1480"}
{attribute addProperty Name "Beckhoff EPP3xxx"}
TYPE Beckhoff_EPP3xxx_37FEE8A0 EXTENDS EK1100_1FC0878B :
STRUCT
	{attribute addProperty Name "Beckhoff EPP3xxxEK1122"}
	{attribute addProperty PreviousPort "Beckhoff EPP3xxx : B"}
	Beckhoff_EPP3xxxEK1122 : Beckhoff_EPP3xxxEK1122_A76E71A7;
END_STRUCT
END_TYPE

// ---- DUTs/IO/Topology/Beckhoff_EPP4xxxEK1122_FE2E0BEF.TcDUT
{attribute 'GeneratedUsingTerminal: EK1122-0000-0018'}
{attribute addProperty BoxType "EK1122-0000-0018"}
{attribute addProperty Id "Beckhoff_EPP4xxxsub_EK1100EK1100_1FC0878B2A_0001_EPP4174_0002_0016EPP4174_AB92710E19A_0002_EPP4174_0002_0017EPP4174_AB92710E19A_0003_EPP4314_1002_0016EPP4314_454AD8BA38A_0004_EPP4374_0002_0016EPP4374_A304750F36A_0005_EPP4374_0002_0017EPP4374_A304750F36A_0006_EPP4374_0002_0018EPP4374_A304750F36A_0007_EPP4374_0002_0019EPP4374_A304750F36"}
{attribute addProperty CRC "4264430575"}
{attribute addProperty Size "222"}
{attribute addProperty Name "Beckhoff EPP4xxxEK1122"}
TYPE Beckhoff_EPP4xxxEK1122_FE2E0BEF EXTENDS EK1122_1FC0878B :
STRUCT
	{attribute addProperty Name "Beckhoff EPP4xxxsub EK1100"}
	{attribute addProperty PreviousPort "Beckhoff EPP4xxxEK1122 : D"}
	Beckhoff_EPP4xxxsub_EK1100 : EK1100_1FC0878B;
	{attribute addProperty Name "A_0001(EPP4174-0002-0016)"}
	{attribute addProperty PreviousPort "Beckhoff EPP4xxxsub EK1100 : C"}
	A_0001_EPP4174_0002_0016 : EPP4174_AB92710E;
	{attribute addProperty Name "A_0002(EPP4174-0002-0017)"}
	{attribute addProperty PreviousPort "A_0001(EPP4174-0002-0016) : B"}
	A_0002_EPP4174_0002_0017 : EPP4174_AB92710E;
	{attribute addProperty Name "A_0003(EPP4314-1002-0016)"}
	{attribute addProperty PreviousPort "A_0002(EPP4174-0002-0017) : B"}
	A_0003_EPP4314_1002_0016 : EPP4314_454AD8BA;
	{attribute addProperty Name "A_0004(EPP4374-0002-0016)"}
	{attribute addProperty PreviousPort "A_0003(EPP4314-1002-0016) : B"}
	A_0004_EPP4374_0002_0016 : EPP4374_A304750F;
	{attribute addProperty Name "A_0005(EPP4374-0002-0017)"}
	{attribute addProperty PreviousPort "A_0004(EPP4374-0002-0016) : B"}
	A_0005_EPP4374_0002_0017 : EPP4374_A304750F;
	{attribute addProperty Name "A_0006(EPP4374-0002-0018)"}
	{attribute addProperty PreviousPort "A_0005(EPP4374-0002-0017) : B"}
	A_0006_EPP4374_0002_0018 : EPP4374_A304750F;
	{attribute addProperty Name "A_0007(EPP4374-0002-0019)"}
	{attribute addProperty PreviousPort "A_0006(EPP4374-0002-0018) : B"}
	A_0007_EPP4374_0002_0019 : EPP4374_A304750F;
END_STRUCT
END_TYPE

// ---- DUTs/IO/Topology/Beckhoff_EPP4xxx_F05B7AA2.TcDUT
{attribute 'GeneratedUsingTerminal: EK1100-0000-0018'}
{attribute addProperty BoxType "EK1100-0000-0018"}
{attribute addProperty Id "Beckhoff_EPP4xxxEK1122Beckhoff_EPP4xxxEK1122_FE2E0BEF222"}
{attribute addProperty CRC "4032527010"}
{attribute addProperty Size "222"}
{attribute addProperty Name "Beckhoff EPP4xxx"}
TYPE Beckhoff_EPP4xxx_F05B7AA2 EXTENDS EK1100_1FC0878B :
STRUCT
	{attribute addProperty Name "Beckhoff EPP4xxxEK1122"}
	{attribute addProperty PreviousPort "Beckhoff EPP4xxx : B"}
	Beckhoff_EPP4xxxEK1122 : Beckhoff_EPP4xxxEK1122_FE2E0BEF;
END_STRUCT
END_TYPE

// ---- DUTs/IO/Topology/Beckhoff_EPP5xxxEK1122_EF1F281E.TcDUT
{attribute 'GeneratedUsingTerminal: EK1122-0000-0018'}
{attribute addProperty BoxType "EK1122-0000-0018"}
{attribute addProperty Id "Beckhoff_EPP5xxxsub_EK1100EK1100_1FC0878B2A_0001_EPP5001_0002_0016EPP5001_0B28D08722A_0002_EPP5101_0002_0016EPP5101_87AC78CF32A_0003_EPP5101_0002_0017EPP5101_87AC78CF32A_0004_EPP5101_0011_0016EPP5101_7476E94838A_0005_EPP5101_0011_0017EPP5101_7476E94838A_0006_EPP5101_1002_0016EPP5101_87AC78CF32A_0007_EPP5101_1002_0017EPP5101_87AC78CF32A_0008_EPP5151_0002_0016EPP5151_7476E94838A_0009_EPP5151_0002_0017EPP5151_7476E94838"}
{attribute addProperty CRC "4011796510"}
{attribute addProperty Size "304"}
{attribute addProperty Name "Beckhoff EPP5xxxEK1122"}
TYPE Beckhoff_EPP5xxxEK1122_EF1F281E EXTENDS EK1122_1FC0878B :
STRUCT
	{attribute addProperty Name "Beckhoff EPP5xxxsub EK1100"}
	{attribute addProperty PreviousPort "Beckhoff EPP5xxxEK1122 : D"}
	Beckhoff_EPP5xxxsub_EK1100 : EK1100_1FC0878B;
	{attribute addProperty Name "A_0001(EPP5001-0002-0016)"}
	{attribute addProperty PreviousPort "Beckhoff EPP5xxxsub EK1100 : C"}
	A_0001_EPP5001_0002_0016 : EPP5001_0B28D087;
	{attribute addProperty Name "A_0002(EPP5101-0002-0016)"}
	{attribute addProperty PreviousPort "A_0001(EPP5001-0002-0016) : B"}
	A_0002_EPP5101_0002_0016 : EPP5101_87AC78CF;
	{attribute addProperty Name "A_0003(EPP5101-0002-0017)"}
	{attribute addProperty PreviousPort "A_0002(EPP5101-0002-0016) : B"}
	A_0003_EPP5101_0002_0017 : EPP5101_87AC78CF;
	{attribute addProperty Name "A_0004(EPP5101-0011-0016)"}
	{attribute addProperty PreviousPort "A_0003(EPP5101-0002-0017) : B"}
	A_0004_EPP5101_0011_0016 : EPP5101_7476E948;
	{attribute addProperty Name "A_0005(EPP5101-0011-0017)"}
	{attribute addProperty PreviousPort "A_0004(EPP5101-0011-0016) : B"}
	A_0005_EPP5101_0011_0017 : EPP5101_7476E948;
	{attribute addProperty Name "A_0006(EPP5101-1002-0016)"}
	{attribute addProperty PreviousPort "A_0005(EPP5101-0011-0017) : B"}
	A_0006_EPP5101_1002_0016 : EPP5101_87AC78CF;
	{attribute addProperty Name "A_0007(EPP5101-1002-0017)"}
	{attribute addProperty PreviousPort "A_0006(EPP5101-1002-0016) : B"}
	A_0007_EPP5101_1002_0017 : EPP5101_87AC78CF;
	{attribute addProperty Name "A_0008(EPP5151-0002-0016)"}
	{attribute addProperty PreviousPort "A_0007(EPP5101-1002-0017) : B"}
	A_0008_EPP5151_0002_0016 : EPP5151_7476E948;
	{attribute addProperty Name "A_0009(EPP5151-0002-0017)"}
	{attribute addProperty PreviousPort "A_0008(EPP5151-0002-0016) : B"}
	A_0009_EPP5151_0002_0017 : EPP5151_7476E948;
END_STRUCT
END_TYPE

// ---- DUTs/IO/Topology/Beckhoff_EPP5xxx_CECB1C9F.TcDUT
{attribute 'GeneratedUsingTerminal: EK1100-0000-0018'}
{attribute addProperty BoxType "EK1100-0000-0018"}
{attribute addProperty Id "Beckhoff_EPP5xxxEK1122Beckhoff_EPP5xxxEK1122_EF1F281E304"}
{attribute addProperty CRC "3469417631"}
{attribute addProperty Size "304"}
{attribute addProperty Name "Beckhoff EPP5xxx"}
TYPE Beckhoff_EPP5xxx_CECB1C9F EXTENDS EK1100_1FC0878B :
STRUCT
	{attribute addProperty Name "Beckhoff EPP5xxxEK1122"}
	{attribute addProperty PreviousPort "Beckhoff EPP5xxx : B"}
	Beckhoff_EPP5xxxEK1122 : Beckhoff_EPP5xxxEK1122_EF1F281E;
END_STRUCT
END_TYPE

// ---- DUTs/IO/Topology/Beckhoff_EPP6xxxEK1122_484AACC3.TcDUT
{attribute 'GeneratedUsingTerminal: EK1122-0000-0018'}
{attribute addProperty BoxType "EK1122-0000-0018"}
{attribute addProperty Id "Beckhoff_EPP6xxxsub_EK1100EK1100_1FC0878B2A_0001_EPP6001_0002_0016EPP6001_40883D0360A_0002_EPP6001_0002_0017EPP6001_40883D0360A_0003_EPP6001_0002_0018EPP6001_40883D0360A_0004_EPP6002_0002_0016EPP6002_7F53816A108A_0005_EPP6002_0002_0017EPP6002_7F53816A108A_0006_EPP6002_0002_0018EPP6002_7BE6B617108A_0007_EPP6002_0002_0019EPP6002_7BE6B617108A_0008_EPP6090_0000_0017EPP6090_18BD01E922A_0009_EPP6228_0022_0016EPP6228_495B58F436"}
{attribute addProperty CRC "1212853443"}
{attribute addProperty Size "672"}
{attribute addProperty Name "Beckhoff EPP6xxxEK1122"}
TYPE Beckhoff_EPP6xxxEK1122_484AACC3 EXTENDS EK1122_1FC0878B :
STRUCT
	{attribute addProperty Name "Beckhoff EPP6xxxsub EK1100"}
	{attribute addProperty PreviousPort "Beckhoff EPP6xxxEK1122 : D"}
	Beckhoff_EPP6xxxsub_EK1100 : EK1100_1FC0878B;
	{attribute addProperty Name "A_0001(EPP6001-0002-0016)"}
	{attribute addProperty PreviousPort "Beckhoff EPP6xxxsub EK1100 : C"}
	A_0001_EPP6001_0002_0016 : EPP6001_40883D03;
	{attribute addProperty Name "A_0002(EPP6001-0002-0017)"}
	{attribute addProperty PreviousPort "A_0001(EPP6001-0002-0016) : B"}
	A_0002_EPP6001_0002_0017 : EPP6001_40883D03;
	{attribute addProperty Name "A_0003(EPP6001-0002-0018)"}
	{attribute addProperty PreviousPort "A_0002(EPP6001-0002-0017) : B"}
	A_0003_EPP6001_0002_0018 : EPP6001_40883D03;
	{attribute addProperty Name "A_0004(EPP6002-0002-0016)"}
	{attribute addProperty PreviousPort "A_0003(EPP6001-0002-0018) : B"}
	A_0004_EPP6002_0002_0016 : EPP6002_7F53816A;
	{attribute addProperty Name "A_0005(EPP6002-0002-0017)"}
	{attribute addProperty PreviousPort "A_0004(EPP6002-0002-0016) : B"}
	A_0005_EPP6002_0002_0017 : EPP6002_7F53816A;
	{attribute addProperty Name "A_0006(EPP6002-0002-0018)"}
	{attribute addProperty PreviousPort "A_0005(EPP6002-0002-0017) : B"}
	A_0006_EPP6002_0002_0018 : EPP6002_7BE6B617;
	{attribute addProperty Name "A_0007(EPP6002-0002-0019)"}
	{attribute addProperty PreviousPort "A_0006(EPP6002-0002-0018) : B"}
	A_0007_EPP6002_0002_0019 : EPP6002_7BE6B617;
	{attribute addProperty Name "A_0008(EPP6090-0000-0017)"}
	{attribute addProperty PreviousPort "A_0007(EPP6002-0002-0019) : B"}
	A_0008_EPP6090_0000_0017 : EPP6090_18BD01E9;
	{attribute addProperty Name "A_0009(EPP6228-0022-0016)"}
	{attribute addProperty PreviousPort "A_0008(EPP6090-0000-0017) : B"}
	A_0009_EPP6228_0022_0016 : EPP6228_495B58F4;
END_STRUCT
END_TYPE

// ---- DUTs/IO/Topology/Beckhoff_EPP6xxx_4A538F0B.TcDUT
{attribute 'GeneratedUsingTerminal: EK1100-0000-0018'}
{attribute addProperty BoxType "EK1100-0000-0018"}
{attribute addProperty Id "Beckhoff_EPP6xxxEK1122Beckhoff_EPP6xxxEK1122_484AACC3672"}
{attribute addProperty CRC "1246990091"}
{attribute addProperty Size "672"}
{attribute addProperty Name "Beckhoff EPP6xxx"}
TYPE Beckhoff_EPP6xxx_4A538F0B EXTENDS EK1100_1FC0878B :
STRUCT
	{attribute addProperty Name "Beckhoff EPP6xxxEK1122"}
	{attribute addProperty PreviousPort "Beckhoff EPP6xxx : B"}
	Beckhoff_EPP6xxxEK1122 : Beckhoff_EPP6xxxEK1122_484AACC3;
END_STRUCT
END_TYPE

// ---- DUTs/IO/Topology/Beckhoff_EPP7xxxEK1122_4AE68EFB.TcDUT
{attribute 'GeneratedUsingTerminal: EK1122-0000-0018'}
{attribute addProperty BoxType "EK1122-0000-0018"}
{attribute addProperty Id "Beckhoff_EPP7xxxsub_EK1100EK1100_1FC0878B2A_0001_EPP7041_1002_0016EPP7041_3210CF4053A_0002_EPP7041_1002_0017EPP7041_3210CF4053A_0003_EPP7041_1002_0023EPP7041_3E4BEAEF54A_0004_EPP7041_3002_0016EPP7041_3E4BEAEF54A_0005_EPP7041_3002_0017EPP7041_3E4BEAEF54A_0006_EPP7041_3002_0018EPP7041_3E4BEAEF54A_0007_EPP7041_3002_0023EPP7041_3E4BEAEF54A_0008_EPP7342_0002_0016EPP7342_2AE9C6B386A_0009_EPP7342_0002_0017EPP7342_2AE9C6B386"}
{attribute addProperty CRC "1256623867"}
{attribute addProperty Size "550"}
{attribute addProperty Name "Beckhoff EPP7xxxEK1122"}
TYPE Beckhoff_EPP7xxxEK1122_4AE68EFB EXTENDS EK1122_1FC0878B :
STRUCT
	{attribute addProperty Name "Beckhoff EPP7xxxsub EK1100"}
	{attribute addProperty PreviousPort "Beckhoff EPP7xxxEK1122 : D"}
	Beckhoff_EPP7xxxsub_EK1100 : EK1100_1FC0878B;
	{attribute addProperty Name "A_0001(EPP7041-1002-0016)"}
	{attribute addProperty PreviousPort "Beckhoff EPP7xxxsub EK1100 : C"}
	A_0001_EPP7041_1002_0016 : EPP7041_3210CF40;
	{attribute addProperty Name "A_0002(EPP7041-1002-0017)"}
	{attribute addProperty PreviousPort "A_0001(EPP7041-1002-0016) : B"}
	A_0002_EPP7041_1002_0017 : EPP7041_3210CF40;
	{attribute addProperty Name "A_0003(EPP7041-1002-0023)"}
	{attribute addProperty PreviousPort "A_0002(EPP7041-1002-0017) : B"}
	A_0003_EPP7041_1002_0023 : EPP7041_3E4BEAEF;
	{attribute addProperty Name "A_0004(EPP7041-3002-0016)"}
	{attribute addProperty PreviousPort "A_0003(EPP7041-1002-0023) : B"}
	A_0004_EPP7041_3002_0016 : EPP7041_3E4BEAEF;
	{attribute addProperty Name "A_0005(EPP7041-3002-0017)"}
	{attribute addProperty PreviousPort "A_0004(EPP7041-3002-0016) : B"}
	A_0005_EPP7041_3002_0017 : EPP7041_3E4BEAEF;
	{attribute addProperty Name "A_0006(EPP7041-3002-0018)"}
	{attribute addProperty PreviousPort "A_0005(EPP7041-3002-0017) : B"}
	A_0006_EPP7041_3002_0018 : EPP7041_3E4BEAEF;
	{attribute addProperty Name "A_0007(EPP7041-3002-0023)"}
	{attribute addProperty PreviousPort "A_0006(EPP7041-3002-0018) : B"}
	A_0007_EPP7041_3002_0023 : EPP7041_3E4BEAEF;
	{attribute addProperty Name "A_0008(EPP7342-0002-0016)"}
	{attribute addProperty PreviousPort "A_0007(EPP7041-3002-0023) : B"}
	A_0008_EPP7342_0002_0016 : EPP7342_2AE9C6B3;
	{attribute addProperty Name "A_0009(EPP7342-0002-0017)"}
	{attribute addProperty PreviousPort "A_0008(EPP7342-0002-0016) : B"}
	A_0009_EPP7342_0002_0017 : EPP7342_2AE9C6B3;
END_STRUCT
END_TYPE

// ---- DUTs/IO/Topology/Beckhoff_EPP7xxx_26C654D6.TcDUT
{attribute 'GeneratedUsingTerminal: EK1100-0000-0018'}
{attribute addProperty BoxType "EK1100-0000-0018"}
{attribute addProperty Id "Beckhoff_EPP7xxxEK1122Beckhoff_EPP7xxxEK1122_4AE68EFB550"}
{attribute addProperty CRC "650532054"}
{attribute addProperty Size "550"}
{attribute addProperty Name "Beckhoff EPP7xxx"}
TYPE Beckhoff_EPP7xxx_26C654D6 EXTENDS EK1100_1FC0878B :
STRUCT
	{attribute addProperty Name "Beckhoff EPP7xxxEK1122"}
	{attribute addProperty PreviousPort "Beckhoff EPP7xxx : B"}
	Beckhoff_EPP7xxxEK1122 : Beckhoff_EPP7xxxEK1122_4AE68EFB;
END_STRUCT
END_TYPE

// ---- DUTs/IO/Topology/Beckhoff_EPP9xxxEK1122_B72DCE23.TcDUT
{attribute 'GeneratedUsingTerminal: EK1122-0000-0018'}
{attribute addProperty BoxType "EK1122-0000-0018"}
{attribute addProperty Id "Beckhoff_EPP9xxxsub_EK1100EK1100_1FC0878B2A_0001_EPP9001_0060_0016EPP9001_1FC0878B2A_0002_EPP9001_0060_0017EPP9001_1FC0878B2A_0003_EPP9022_0060_0017EPP9022_32A9C19F48A_0004_EPP9022_9060_0017EPP9022_32A9C19F48"}
{attribute addProperty CRC "3073232419"}
{attribute addProperty Size "102"}
{attribute addProperty Name "Beckhoff EPP9xxxEK1122"}
TYPE Beckhoff_EPP9xxxEK1122_B72DCE23 EXTENDS EK1122_1FC0878B :
STRUCT
	{attribute addProperty Name "Beckhoff EPP9xxxsub EK1100"}
	{attribute addProperty PreviousPort "Beckhoff EPP9xxxEK1122 : D"}
	Beckhoff_EPP9xxxsub_EK1100 : EK1100_1FC0878B;
	{attribute addProperty Name "A_0001(EPP9001-0060-0016)"}
	{attribute addProperty PreviousPort "Beckhoff EPP9xxxsub EK1100 : C"}
	A_0001_EPP9001_0060_0016 : EPP9001_1FC0878B;
	{attribute addProperty Name "A_0002(EPP9001-0060-0017)"}
	{attribute addProperty PreviousPort "A_0001(EPP9001-0060-0016) : B"}
	A_0002_EPP9001_0060_0017 : EPP9001_1FC0878B;
	{attribute addProperty Name "A_0003(EPP9022-0060-0017)"}
	{attribute addProperty PreviousPort "A_0002(EPP9001-0060-0017) : B"}
	A_0003_EPP9022_0060_0017 : EPP9022_32A9C19F;
	{attribute addProperty Name "A_0004(EPP9022-9060-0017)"}
	{attribute addProperty PreviousPort "A_0003(EPP9022-0060-0017) : B"}
	A_0004_EPP9022_9060_0017 : EPP9022_32A9C19F;
END_STRUCT
END_TYPE

// ---- DUTs/IO/Topology/Beckhoff_EPP9xxx_3F2579D7.TcDUT
{attribute 'GeneratedUsingTerminal: EK1100-0000-0018'}
{attribute addProperty BoxType "EK1100-0000-0018"}
{attribute addProperty Id "Beckhoff_EPP9xxxEK1122Beckhoff_EPP9xxxEK1122_B72DCE23102"}
{attribute addProperty CRC "1059420631"}
{attribute addProperty Size "102"}
{attribute addProperty Name "Beckhoff EPP9xxx"}
TYPE Beckhoff_EPP9xxx_3F2579D7 EXTENDS EK1100_1FC0878B :
STRUCT
	{attribute addProperty Name "Beckhoff EPP9xxxEK1122"}
	{attribute addProperty PreviousPort "Beckhoff EPP9xxx : B"}
	Beckhoff_EPP9xxxEK1122 : Beckhoff_EPP9xxxEK1122_B72DCE23;
END_STRUCT
END_TYPE

// ---- DUTs/IO/Topology/EtherCAT_Master_EPPxxxx_9A8F5D7B.TcDUT
{attribute 'GeneratedUsingTerminal: IODEVICETYPE_ETHERCATPROT'}
{attribute addProperty BoxType "IODEVICETYPE_ETHERCATPROT"}
{attribute addProperty Id "Beckhoff_EPP1xxxBeckhoff_EPP1xxx_3250354D762Beckhoff_EPP2xxxBeckhoff_EPP2xxx_8ED37E642100Beckhoff_EPP3xxxBeckhoff_EPP3xxx_37FEE8A01480Beckhoff_EPP4xxxBeckhoff_EPP4xxx_F05B7AA2222Beckhoff_EPP5xxxBeckhoff_EPP5xxx_CECB1C9F304Beckhoff_EPP6xxxBeckhoff_EPP6xxx_4A538F0B672Beckhoff_EPP7xxxBeckhoff_EPP7xxx_26C654D6550Beckhoff_EPP9xxxBeckhoff_EPP9xxx_3F2579D7102SyncUnitsSyncUnits_99E584AF18InputsInputs_25A0042B160OutputsOutputs_2397A10E106InfoDataInfoData_E68C61CD28"}
{attribute addProperty CRC "2593086843"}
{attribute addProperty Size "6504"}
{attribute addProperty Name "EtherCAT Master EPPxxxx"}
TYPE EtherCAT_Master_EPPxxxx_9A8F5D7B EXTENDS EtcMasterBase_62654B43 :
STRUCT
	{attribute addProperty Name "Beckhoff EPP1xxx"}
	{attribute addProperty PreviousPort "EtherCAT Master EPPxxxx : Master"}
	Beckhoff_EPP1xxx : Beckhoff_EPP1xxx_3250354D;
	{attribute addProperty Name "Beckhoff EPP2xxx"}
	{attribute addProperty PreviousPort "Beckhoff EPP1xxx : C"}
	Beckhoff_EPP2xxx : Beckhoff_EPP2xxx_8ED37E64;
	{attribute addProperty Name "Beckhoff EPP3xxx"}
	{attribute addProperty PreviousPort "Beckhoff EPP2xxx : C"}
	Beckhoff_EPP3xxx : Beckhoff_EPP3xxx_37FEE8A0;
	{attribute addProperty Name "Beckhoff EPP4xxx"}
	{attribute addProperty PreviousPort "Beckhoff EPP3xxx : C"}
	Beckhoff_EPP4xxx : Beckhoff_EPP4xxx_F05B7AA2;
	{attribute addProperty Name "Beckhoff EPP5xxx"}
	{attribute addProperty PreviousPort "Beckhoff EPP4xxx : C"}
	Beckhoff_EPP5xxx : Beckhoff_EPP5xxx_CECB1C9F;
	{attribute addProperty Name "Beckhoff EPP6xxx"}
	{attribute addProperty PreviousPort "Beckhoff EPP5xxx : C"}
	Beckhoff_EPP6xxx : Beckhoff_EPP6xxx_4A538F0B;
	{attribute addProperty Name "Beckhoff EPP7xxx"}
	{attribute addProperty PreviousPort "Beckhoff EPP6xxx : C"}
	Beckhoff_EPP7xxx : Beckhoff_EPP7xxx_26C654D6;
	{attribute addProperty Name "Beckhoff EPP9xxx"}
	{attribute addProperty PreviousPort "Beckhoff EPP7xxx : C"}
	Beckhoff_EPP9xxx : Beckhoff_EPP9xxx_3F2579D7;
	{attribute addProperty Name "SyncUnits"}
	SyncUnits : SyncUnits_99E584AF;
	{attribute addProperty Name "Inputs"}
	Inputs : Inputs_25A0042B;
	{attribute addProperty Name "Outputs"}
	Outputs : Outputs_2397A10E;
	{attribute addProperty Name "InfoData"}
	InfoData : InfoData_E68C61CD;
END_STRUCT
END_TYPE

// ---- DUTs/IO/Base/EtcSlaveBase_82538BE2.TcDUT

TYPE EtcSlaveBase_82538BE2 :
STRUCT
END_STRUCT
END_TYPE

// ---- DUTs/IO/Base/EtcSlaveBase_82538BE2.TcDUT

TYPE EtcSlaveBase_82538BE2 :
STRUCT
END_STRUCT
END_TYPE

// ---- DUTs/IO/Base/EtcSlaveBase_82538BE2.TcDUT

TYPE EtcSlaveBase_82538BE2 :
STRUCT
END_STRUCT
END_TYPE

// ---- DUTs/IO/Base/EtcSlaveTerminalBase_947E5A46.TcDUT

{attribute clr[Container(Layout.Stack)]}
{attribute clr[Group(Layout.GroupBox)]}
{attribute addProperty PreviousPort "Unknown"}
TYPE EtcSlaveTerminalBase_947E5A46 EXTENDS EtcSlaveBase_82538BE2 :
STRUCT
END_STRUCT
END_TYPE

// ---- DUTs/IO/Base/EtcSlaveBoxBase_77A0E4A7.TcDUT

{attribute clr[Container(Layout.Stack)]}
{attribute clr[Group(Layout.GroupBox)]}
{attribute addProperty PreviousPort "Unknown"}
TYPE EtcSlaveBoxBase_77A0E4A7 EXTENDS EtcSlaveBase_82538BE2 :
STRUCT
END_STRUCT
END_TYPE

// ---- DUTs/IO/Base/EtcSlaveEndTerminalBase_866C7F0C.TcDUT

{attribute clr[Container(Layout.Stack)]}
{attribute clr[Group(Layout.GroupBox)]}
{attribute addProperty PreviousPort "Unknown"}
TYPE EtcSlaveEndTerminalBase_866C7F0C EXTENDS EtcSlaveBase_82538BE2 :
STRUCT
END_STRUCT
END_TYPE

// ---- DUTs/IO/Base/InputBase_8311D824.TcDUT

TYPE InputBase_8311D824 :
STRUCT
END_STRUCT
END_TYPE

// ---- DUTs/IO/Base/OutputBase_10CEE7DE.TcDUT

TYPE OutputBase_10CEE7DE :
STRUCT
END_STRUCT
END_TYPE

// ---- DUTs/IO/Base/EtcMasterBase_62654B43.TcDUT

TYPE EtcMasterBase_62654B43 :
STRUCT
END_STRUCT
END_TYPE

// ---- GVLs/GVL_iXlinker.TcGVL
{attribute 'qualified_only'}
VAR_GLOBAL
		EtherCAT_Master_EPPxxxx : EtherCAT_Master_EPPxxxx_9A8F5D7B;
END_VAR

// ---- POUs/MAIN.TcPOU
PROGRAM MAIN
VAR
END_VAR

END_PROGRAM
